TYPE STRUCT_ModeSelect :
STRUCT
	Auto	: BOOL;
	Manueel	: BOOL;
	Tag		: STRING;
END_STRUCT
END_TYPE

(* stored: Version 1.1.0.1, ProductVersion 3.1.4024.12
   DUT STRUCT_ModeSelect: Id {61212d08-0fe2-48f3-b858-5e96aefbf3e1} *)
